FUNCTION_BLOCK _ETcVnBorderInterpolationMethod_TestSuite EXTENDS TcUnit.FB_TestSuite
VAR
END_VAR

TestAddress();
TestClearReference();
TestClone();
TestTypeNameReturnsExpected();
TestIdentifierReturnsExpected();
TestMakeReferenceToFollowsReference();
TestMakeReferenceToUpdatesReference();
TestSize();
TestValueReturnsExpectedAfterInit();
TestValueReturnsExpectedAfterChange();
TestSerializeTypeWith();
TestSerializeWith();
TestTryDeserializeFrom();
TestTryMakeReferenceToFollowsReference();
TestTryMakeReferenceToUpdatesReference();

METHOD PUBLIC TestAddress
VAR
    _type : _ETcVnBorderInterpolationMethod(ETcVnBorderInterpolationMethod.TCVN_BIM_CONSTANT);
    notExpected : PVOID := 0;
    actual : PVOID;
END_VAR
TEST('TestAddress');

actual := _type.Address;

AssertFalse(
    Condition := (notExpected = actual),
    Message := 'Type did not return a valid address.'
);

TEST_FINISHED();
END_METHOD

METHOD PUBLIC TestClearReference
VAR
    _type : _ETcVnBorderInterpolationMethod(ETcVnBorderInterpolationMethod.TCVN_BIM_CONSTANT);
	target : ETcVnBorderInterpolationMethod := ETcVnBorderInterpolationMethod.TCVN_BIM_CONSTANT;
    expected : ETcVnBorderInterpolationMethod := ETcVnBorderInterpolationMethod.TCVN_BIM_CONSTANT;
    actual : ETcVnBorderInterpolationMethod;
END_VAR
TEST('TestClearReference');

_type.MakeReferenceTo(target);
_type.ClearReference();
target := ETcVnBorderInterpolationMethod.TCVN_BIM_REPLICATE;

actual := _type.Value;

AssertEquals(
    Expected := expected,
    Actual := actual,
    Message := 'Value continued to follow target.'
);

TEST_FINISHED();
END_METHOD

METHOD PUBLIC TestClone
VAR
    _type : _ETcVnBorderInterpolationMethod(ETcVnBorderInterpolationMethod.TCVN_BIM_CONSTANT);
	clone : I_Datatype;
	isValidClone : BOOL;
	compareResult : DINT;
END_VAR
TEST('TestClone');

clone := _type.Clone();

isValidClone := clone <> 0;

IF isValidClone THEN
	compareResult := memcmp(_type.Address, clone.Address, clone.Size);
END_IF

AssertTrue(
	Condition := isValidClone,
	Message := 'Clone did not produce a clone'
);

AssertEquals_DINT(
	Expected := 0,
    Actual := compareResult,
    Message := 'Clone did not return a valid clone.'
);

clone.Dispose();

TEST_FINISHED();
END_METHOD

METHOD PUBLIC TestIdentifierReturnsExpected
VAR
    _type : _ETcVnBorderInterpolationMethod(ETcVnBorderInterpolationMethod.TCVN_BIM_CONSTANT);
    expected : STRING := 'ETcVnBorderInterpolationMethod';
    actual : STRING;
END_VAR
TEST('TestIdentifierReturnsExpected');

actual := _type.Identifier;

AssertEquals_STRING(
    Expected := expected,
    Actual := actual,
    Message := 'Type did not return correct iec type.'
);

TEST_FINISHED();
END_METHOD

METHOD PUBLIC TestMakeReferenceToFollowsReference
VAR
    _type : _ETcVnBorderInterpolationMethod(ETcVnBorderInterpolationMethod.TCVN_BIM_CONSTANT);
	target : ETcVnBorderInterpolationMethod := ETcVnBorderInterpolationMethod.TCVN_BIM_CONSTANT;
    expected : ETcVnBorderInterpolationMethod := ETcVnBorderInterpolationMethod.TCVN_BIM_REPLICATE;
    actual : ETcVnBorderInterpolationMethod;
END_VAR
TEST('TestMakeReferenceToFollowsReference');

_type.MakeReferenceTo(target);
target := ETcVnBorderInterpolationMethod.TCVN_BIM_REPLICATE;

actual := _type.Value;

AssertEquals(
    Expected := expected,
    Actual := actual,
    Message := 'Value did not follow target change.'
);

TEST_FINISHED();
END_METHOD

METHOD PUBLIC TestMakeReferenceToUpdatesReference
VAR
    _type : _ETcVnBorderInterpolationMethod(ETcVnBorderInterpolationMethod.TCVN_BIM_CONSTANT);
	target : ETcVnBorderInterpolationMethod := ETcVnBorderInterpolationMethod.TCVN_BIM_CONSTANT;
    expected : ETcVnBorderInterpolationMethod := ETcVnBorderInterpolationMethod.TCVN_BIM_REPLICATE;
    actual : ETcVnBorderInterpolationMethod;
END_VAR
TEST('TestMakeReferenceToUpdatesReference');

_type.MakeReferenceTo(target);
_type.Value := ETcVnBorderInterpolationMethod.TCVN_BIM_REPLICATE;

actual := target;

AssertEquals(
    Expected := expected,
    Actual := actual,
    Message := 'Value did not update target.'
);

TEST_FINISHED();
END_METHOD

METHOD PUBLIC TestSerializeTypeWith
VAR
    _type : _ETcVnBorderInterpolationMethod(ETcVnBorderInterpolationMethod.TCVN_BIM_CONSTANT);
    serializer : JsonSerializer;
    expected : STRING(500) := '{"typeName":"ENUM","identifier":"ETcVnBorderInterpolationMethod","enumerations":["TCVN_BIM_CONSTANT","TCVN_BIM_REPLICATE","TCVN_BIM_REFLECT","TCVN_BIM_WRAP","TCVN_BIM_REFLECT_101","TCVN_BIM_DEFAULT","TCVN_BIM_TRANSPARENT","TCVN_BIM_ISOLATED_CONSTANT","TCVN_BIM_ISOLATED_REPLICATE","TCVN_BIM_ISOLATED_REFLECT","TCVN_BIM_ISOLATED_WRAP","TCVN_BIM_ISOLATED_REFLECT_101"],"baseType":{"typeName":"DINT","minValue":-2147483648,"maxValue":2147483647,"isSigned":true,"isFloat":false}}'; 
    actual : STRING(500);
END_VAR
TEST('TestSerializeTypeWith');

serializer.Reset();
_type.SerializeTypeWith(serializer);
serializer.TryGetSerializedData(ADR(actual), SIZEOF(actual));

AssertEquals_STRING(
    Expected := expected,
    Actual := actual,
    Message := 'Serialization of type did not return correct string.'
);

TEST_FINISHED();
END_METHOD

METHOD PUBLIC TestSerializeWith
VAR
    _type : _ETcVnBorderInterpolationMethod(ETcVnBorderInterpolationMethod.TCVN_BIM_CONSTANT);
    serializer : JsonSerializer;
    expected : STRING := '"TCVN_BIM_CONSTANT"';
    actual : STRING(500);
END_VAR
TEST('TestSerializeWith');

serializer.Reset();
_type.SerializeWith(serializer);
serializer.TryGetSerializedData(ADR(actual), SIZEOF(actual));

AssertEquals_STRING(
    Expected := expected,
    Actual := actual,
    Message := 'Serialization of type data did not return correct string.'
);

TEST_FINISHED();
END_METHOD

METHOD PUBLIC TestSize
VAR
    _type : _ETcVnBorderInterpolationMethod(ETcVnBorderInterpolationMethod.TCVN_BIM_CONSTANT);
    expected : UDINT := SIZEOF(ETcVnBorderInterpolationMethod);
    actual : UDINT;
END_VAR
TEST('TestSize');

actual := _type.Size;

AssertEquals_UDINT(
    Expected := Expected,
    Actual := actual,
    Message := 'Type did not return the correct size.'
);

TEST_FINISHED();
END_METHOD

METHOD PUBLIC TestTryDeserializeFrom
VAR
    deserializer : JsonDeserializer;
    feedback : DeserializerFeedback;
    json : STRING := '"TCVN_BIM_CONSTANT"';
    _type : _ETcVnBorderInterpolationMethod(ETcVnBorderInterpolationMethod.TCVN_BIM_CONSTANT);
    expected : ETcVnBorderInterpolationMethod := ETcVnBorderInterpolationMethod.TCVN_BIM_CONSTANT;
    actual : ETcVnBorderInterpolationMethod;
 END_VAR
TEST('TestTryDeserializeFrom');

deserializer.Reset();
deserializer.TryLoad(json);
_type.TryDeserializeFrom(Deserializer, Feedback);

actual := _type.Value;

AssertEquals(
    Expected := expected,
    Actual := actual,
    Message := 'Type did not deserialize correctly.'
);

TEST_FINISHED();
END_METHOD

METHOD PUBLIC TestTryMakeReferenceToFollowsReference
VAR
    _type : _ETcVnBorderInterpolationMethod(ETcVnBorderInterpolationMethod.TCVN_BIM_CONSTANT);
	target : _ETcVnBorderInterpolationMethod(ETcVnBorderInterpolationMethod.TCVN_BIM_CONSTANT);
    expected : ETcVnBorderInterpolationMethod := ETcVnBorderInterpolationMethod.TCVN_BIM_REPLICATE;
    actual : ETcVnBorderInterpolationMethod;
END_VAR
TEST('TestTryMakeReferenceToFollowsReference');

_type.TryMakeReferenceTo(target);
target.Value := ETcVnBorderInterpolationMethod.TCVN_BIM_REPLICATE;

actual := _type.Value;

AssertEquals(
    Expected := expected,
    Actual := actual,
    Message := 'Value did not follow target change.'
);

TEST_FINISHED();
END_METHOD

METHOD PUBLIC TestTryMakeReferenceToUpdatesReference
VAR
    _type : _ETcVnBorderInterpolationMethod(ETcVnBorderInterpolationMethod.TCVN_BIM_CONSTANT);
	target : _ETcVnBorderInterpolationMethod(ETcVnBorderInterpolationMethod.TCVN_BIM_CONSTANT);
    expected : ETcVnBorderInterpolationMethod := ETcVnBorderInterpolationMethod.TCVN_BIM_REPLICATE;
    actual : ETcVnBorderInterpolationMethod;
END_VAR
TEST('TestTryMakeReferenceToUpdatesReference');

_type.TryMakeReferenceTo(target);
_type.Value := ETcVnBorderInterpolationMethod.TCVN_BIM_REPLICATE;

actual := target.Value;

AssertEquals(
    Expected := expected,
    Actual := actual,
    Message := 'Value did not update target.'
);

TEST_FINISHED();
END_METHOD

METHOD PUBLIC TestTypeNameReturnsExpected
VAR
    _type : _ETcVnBorderInterpolationMethod(ETcVnBorderInterpolationMethod.TCVN_BIM_CONSTANT);
    expected : STRING := 'ENUM';
    actual : STRING;
END_VAR
TEST('TestTypeNameReturnsExpected');

actual := _type.TypeName;

AssertEquals_STRING(
    Expected := expected,
    Actual := actual,
    Message := 'Type did not return correct iec type.'
);

TEST_FINISHED();
END_METHOD

METHOD PUBLIC TestValueReturnsExpectedAfterChange
VAR
    _type : _ETcVnBorderInterpolationMethod(ETcVnBorderInterpolationMethod.TCVN_BIM_CONSTANT);
    expected : ETcVnBorderInterpolationMethod := ETcVnBorderInterpolationMethod.TCVN_BIM_REPLICATE;
    actual : ETcVnBorderInterpolationMethod;
END_VAR
TEST('TestValueReturnsExpectedAfterChange');

_type.Value := ETcVnBorderInterpolationMethod.TCVN_BIM_REPLICATE;

actual := _type.Value;

AssertEquals(
    Expected := expected,
    Actual := actual,
    Message := 'Expected value not returned after change.'
);

TEST_FINISHED();
END_METHOD

METHOD PUBLIC TestValueReturnsExpectedAfterInit
VAR
    _type : _ETcVnBorderInterpolationMethod(ETcVnBorderInterpolationMethod.TCVN_BIM_CONSTANT);
    expected : ETcVnBorderInterpolationMethod := ETcVnBorderInterpolationMethod.TCVN_BIM_CONSTANT;
    actual : ETcVnBorderInterpolationMethod;
END_VAR
TEST('TestValueReturnsExpectedAfterInit');

actual := _type.Value;

AssertEquals(
    Expected := expected,
    Actual := actual,
    Message := 'Expected value not returned after Init.'
);

TEST_FINISHED();
END_METHOD

END_FUNCTION_BLOCK

(* stored: Version 1.1.0.1, ProductVersion 3.1.4024.12
   POU _ETcVnBorderInterpolationMethod_TestSuite: Id {5919beff-33e9-0b7a-1ff9-aac8e71afa10}, SpecialFunc None
   Method TestAddress: Id {043aa420-7244-0e8f-0f8c-d6088d07d009}
   Method TestClearReference: Id {a528a3dd-e2cc-0117-0e7c-2e592e360e78}
   Method TestClone: Id {fb7d18d6-ec9e-0249-06d7-b630fc19a1ca}
   Method TestIdentifierReturnsExpected: Id {38d80106-10a0-0d00-0f1a-597932eee25c}
   Method TestMakeReferenceToFollowsReference: Id {abda4f6d-ec72-0d2a-12d0-497cd752e453}
   Method TestMakeReferenceToUpdatesReference: Id {0030248f-49cd-0a72-0a23-dc31969fef26}
   Method TestSerializeTypeWith: Id {a611467c-19fa-0284-03d9-8dada5a76db2}
   Method TestSerializeWith: Id {0f6a2de0-54ab-001f-0aec-3164319af1ad}
   Method TestSize: Id {c418b1fe-e4a6-0d70-0103-46fcd537485f}
   Method TestTryDeserializeFrom: Id {4a616fca-f938-0d97-0122-eeb17a0eecd5}
   Method TestTryMakeReferenceToFollowsReference: Id {f9c7a5d2-ba74-07d3-0b42-8836aa45f50f}
   Method TestTryMakeReferenceToUpdatesReference: Id {aeddf891-e913-0a2f-1e9e-7af5fc2d0f77}
   Method TestTypeNameReturnsExpected: Id {fb93e855-a9e5-087b-3fa1-7625f9e572dc}
   Method TestValueReturnsExpectedAfterChange: Id {163cfa6b-b92f-09ed-0e38-e57cf737ef06}
   Method TestValueReturnsExpectedAfterInit: Id {a22b98e4-da67-0345-22ae-3bc6c864df84} *)
